FUNCTION_BLOCK FB_Boolean
VAR_INPUT
    bInput  : BOOL;
END_VAR
VAR_OUTPUT
    bResult : BOOL;
END_VAR

bResult := NOT bInput;

END_FUNCTION_BLOCK

(* stored: Version 1.1.0.1, ProductVersion 3.1.4024.10
   POU FB_Boolean: KindOfPOU Element *)
